TYPE E_SYSTEM_CTState :
(
	E_SYSTEMCT_IDLE,
	E_SYSTEMCT_TIMEZONE,
	E_SYSTEMCT_SYSTEMTIME,
	E_SYSTEMCT_SETSYSTEMTIME,
	E_SYSTEMCT_ERROR,
	E_SYSTEMCT_CREATETEMPFOLDER,
	E_SYSTEMCT_CREATEBASEFOLDER,
	E_SYSTEMCT_DONE
);
END_TYPE

(* stored: Version 1.1.0.1, ProductVersion 3.1.4024.15
   DUT E_SYSTEM_CTState: Id {6815fcf3-4731-49b7-8fdc-ffe73c751e2d} *)
